// TIA Portal V20 export
// export: Created 2026-07-10T11:12:24.5960656Z, ExportSetting WithDefaults, DisplayName Totally Integrated Automation Portal, DisplayVersion V20, DisplayName TIA Portal Openness, DisplayVersion V20, DisplayName TIA Portal Version Control Interface, DisplayVersion V20, DisplayName STEP 7 Professional, DisplayVersion V20, DisplayName STEP 7 Safety, DisplayVersion V20, DisplayName WinCC Basic/Comfort/Advanced, DisplayVersion V20, DisplayName WinCC Unified, DisplayVersion V20
FUNCTION_BLOCK "HMI"   // FB16, SCL
{ S7_Optimized_Access := 'TRUE' }
VERSION : 0.1
// stored: AutoNumber true, IsIECCheckEnabled false, IsRetainMemResEnabled false, MemoryReserve 100, SetENOAutomatically false, UDAEnableTagReadback false
   VAR
      UpdateTimer { S7_SetPoint := 'True'} : TON_TIME;
   END_VAR
   VAR_TEMP
      Ret : Int;
   END_VAR
BEGIN
   "Config".HMI_ResetWaterCounter := "MB".Table.HMI_ResetWaterCounter;
   IF "MB".Table.HMI_ResetWaterCounter THEN
       "MB".Table.HMI_ResetWaterCounter := 0;
   END_IF;

   "Config".HMI_ResetPositionDamper1 := "MB".Table.HMI_ResetPositionDamper1;
   IF "MB".Table.HMI_ResetPositionDamper1 THEN
       "MB".Table.HMI_ResetPositionDamper1 := 0;
   END_IF;

   "Config".HMI_ResetPositionDamper2 := "MB".Table.HMI_ResetPositionDamper2;
   IF "MB".Table.HMI_ResetPositionDamper2 THEN
       "MB".Table.HMI_ResetPositionDamper2 := 0;
   END_IF;

   "Config".HMI_StartAdjustDamper1 := "MB".Table.HMI_StartAdjustDamper1;
   IF "MB".Table.HMI_StartAdjustDamper1 THEN
       "MB".Table.HMI_StartAdjustDamper1 := 0;
   END_IF;

   "Config".HMI_StartAdjustDamper2 := "MB".Table.HMI_StartAdjustDamper2;
   IF "MB".Table.HMI_StartAdjustDamper2 THEN
       "MB".Table.HMI_StartAdjustDamper2 := 0;
   END_IF;

   "Config".HMI_StopAdjustDamper1 := "MB".Table.HMI_StopAdjustDamper1;
   IF "MB".Table.HMI_StopAdjustDamper1 THEN
       "MB".Table.HMI_StopAdjustDamper1 := 0;
   END_IF;

   "Config".HMI_StopAdjustDamper2 := "MB".Table.HMI_StopAdjustDamper2;
   IF "MB".Table.HMI_StopAdjustDamper2 THEN
       "MB".Table.HMI_StopAdjustDamper2 := 0;
   END_IF;

   "Config".HMI_WeightToZero := "MB".Table.HMI_WeightToZero;
   IF "MB".Table.HMI_WeightToZero THEN
       "MB".Table.HMI_WeightToZero := 0;
   END_IF;

   IF "MB".Table.ChlorReg_Update THEN
       "MB".Table.ChlorReg_ChlorValueRCV := "MB".Table.HMI_ChlorReg_ValueRCV;
       "MB".Table.ChlorReg_ChlorValuePt := "MB".Table.HMI_ChlorReg_ValuePt;
       "MB".Table.ChlorReg_Age := "MB".Table.CycleDay;
       "MB".Table.ChlorReg_AgeF := INT_TO_REAL("MB".Table.CycleDay);
       #Ret:= RD_SYS_T("MB".Table.ChlorReg_DateTime);
       #UpdateTimer(IN:=TRUE,
                    PT:=T#100ms);
       IF #UpdateTimer.Q THEN
           "MB".Table.ChlorReg_Update := FALSE;
           RESET_TIMER(#UpdateTimer);
       END_IF;


   END_IF;
END_FUNCTION_BLOCK
